// TIA Portal V20 export
FUNCTION_BLOCK "FB_Analogic_Input"   // FB2, LAD
{ S7_Optimized_Access := 'TRUE' }
// Leitura das 2 Entradas Analogica de um CLP S7 1200 1214 DC/DC/DC
// stored: AutoNumber false, IsIECCheckEnabled true, MemoryReserve 100, SetENOAutomatically false
   VAR_INPUT
      Analogic_Input_0 { ExternalAccessible := 'False'; ExternalVisible := 'False'; ExternalWritable := 'False'} : Int;
      Analogic_Input_1 { ExternalAccessible := 'False'; ExternalVisible := 'False'; ExternalWritable := 'False'} : Int;
      Min_NormX_AI_0 { ExternalAccessible := 'False'; ExternalVisible := 'False'; ExternalWritable := 'False'} : Int := 0;
      Max_NormX_AI_0 { ExternalAccessible := 'False'; ExternalVisible := 'False'; ExternalWritable := 'False'} : Int := 27648;
      Min_NormX_AI_1 { ExternalAccessible := 'False'; ExternalVisible := 'False'; ExternalWritable := 'False'} : Int := 0;
      Max_NormX_AI_1 { ExternalAccessible := 'False'; ExternalVisible := 'False'; ExternalWritable := 'False'} : Int := 27648;
      Scale_Min_AI_0 { ExternalAccessible := 'False'; ExternalVisible := 'False'; ExternalWritable := 'False'} : Real;
      Scale_Max_AI_0 { ExternalAccessible := 'False'; ExternalVisible := 'False'; ExternalWritable := 'False'} : Real;
      Scale_Min_AI_1 { ExternalAccessible := 'False'; ExternalVisible := 'False'; ExternalWritable := 'False'} : Real;
      Scale_Max_AI_1 { ExternalAccessible := 'False'; ExternalVisible := 'False'; ExternalWritable := 'False'} : Real;
   END_VAR
   VAR_OUTPUT
      Value_Real_AI_0 { ExternalAccessible := 'False'; ExternalVisible := 'False'; ExternalWritable := 'False'} : Real;
      Value_Real_AI_1 { ExternalAccessible := 'False'; ExternalVisible := 'False'; ExternalWritable := 'False'} : Real;
      Value_UInt_AI_0 : UInt;
      Value_UInt_AI_1 : UInt;
   END_VAR
   VAR
      Norm_X_Out_AI_0 { ExternalAccessible := 'False'; ExternalVisible := 'False'; ExternalWritable := 'False'} : Real;
      Norm_X_Out_AI_1 { ExternalAccessible := 'False'; ExternalVisible := 'False'; ExternalWritable := 'False'} : Real;
   END_VAR
BEGIN

REGION Network 1: Analogic Input 0
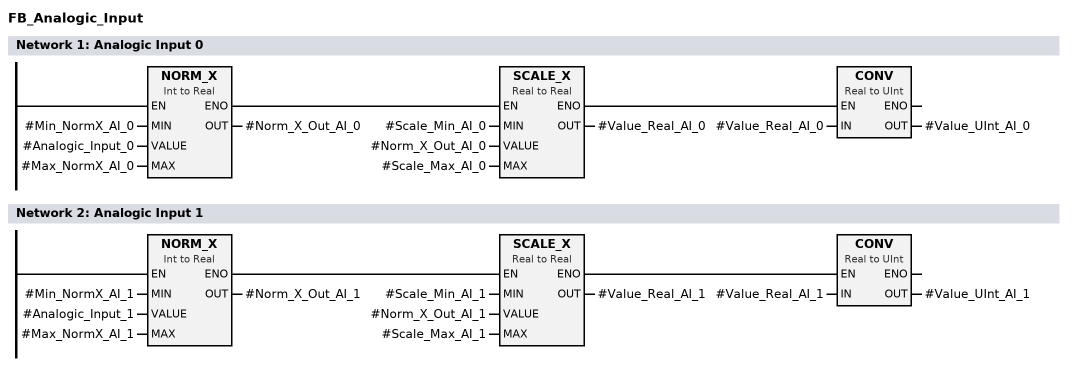
   RUNG wire#powerrail
      { S7_Templates := "[SrcType := Int, DestType := Real]" } Normalize(min := #Min_NormX_AI_0, value := #Analogic_Input_0, max := #Max_NormX_AI_0, out => #Norm_X_Out_AI_0)
      { S7_Templates := "[SrcType := Real, DestType := Real]" } Scale(min := #Scale_Min_AI_0, value := #Norm_X_Out_AI_0, max := #Scale_Max_AI_0, out => #Value_Real_AI_0)
      { S7_Templates := "[SrcType := Real, DestType := UInt]" } Convert(in := #Value_Real_AI_0, out => #Value_UInt_AI_0)
   END_RUNG
   // the same network as SCL:
   #Norm_X_Out_AI_0 := NORM_X(MIN := #Min_NormX_AI_0, VALUE := #Analogic_Input_0, MAX := #Max_NormX_AI_0);
   #Value_Real_AI_0 := SCALE_X(MIN := #Scale_Min_AI_0, VALUE := #Norm_X_Out_AI_0, MAX := #Scale_Max_AI_0);
   #Value_UInt_AI_0 := REAL_TO_UINT(#Value_Real_AI_0);
END_REGION

REGION Network 2: Analogic Input 1
   RUNG wire#powerrail
      { S7_Templates := "[SrcType := Int, DestType := Real]" } Normalize(min := #Min_NormX_AI_1, value := #Analogic_Input_1, max := #Max_NormX_AI_1, out => #Norm_X_Out_AI_1)
      { S7_Templates := "[SrcType := Real, DestType := Real]" } Scale(min := #Scale_Min_AI_1, value := #Norm_X_Out_AI_1, max := #Scale_Max_AI_1, out => #Value_Real_AI_1)
      { S7_Templates := "[SrcType := Real, DestType := UInt]" } Convert(in := #Value_Real_AI_1, out => #Value_UInt_AI_1)
   END_RUNG
   // the same network as SCL:
   #Norm_X_Out_AI_1 := NORM_X(MIN := #Min_NormX_AI_1, VALUE := #Analogic_Input_1, MAX := #Max_NormX_AI_1);
   #Value_Real_AI_1 := SCALE_X(MIN := #Scale_Min_AI_1, VALUE := #Norm_X_Out_AI_1, MAX := #Scale_Max_AI_1);
   #Value_UInt_AI_1 := REAL_TO_UINT(#Value_Real_AI_1);
END_REGION
END_FUNCTION_BLOCK
